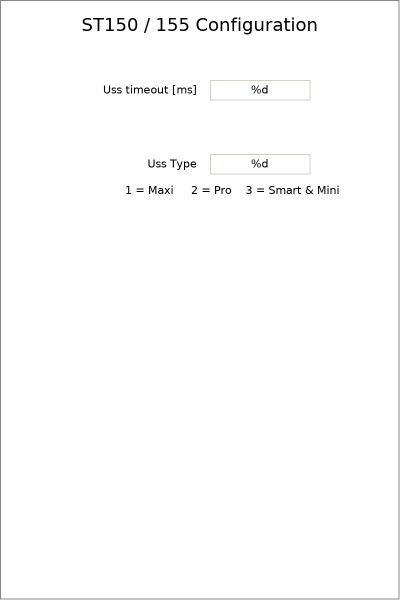
VISUALIZATION VISU_Recipe_ST150  // 400x600
    Textfield (210,80 100x20), "%d", text variable: _20_AUTO.recipe.st150.USS_ErrorTime_ms
        OnMouseDown: write the text variable via Default
    Label (0,5 400x40), "ST150 / 155 Configuration"
    Label (0,80 200x20), "Uss timeout [ms]"
    Textfield (210,154 100x20), "%d", text variable: _20_AUTO.recipe.st150.USS_Type
        OnMouseDown: write the text variable via Default
    Label (0,154 200x20), "Uss Type"
    Label (112,176 241x29), "1 = Maxi 2 = Pro 3 = Smart & Mini"
END_VISUALIZATION

(* stored: Version 1.1.0.1, ProductVersion 3.1.4024.6
   Visu VISU_Recipe_ST150: Id {b7febd48-a0ba-435e-9510-3dc76df45ef3} *)
